// TIA Portal V20 export
DATA_BLOCK "instFB_AxisCtrl"   // DB
TITLE = Axis Control instance DB
{ S7_Optimized_Access := 'TRUE' }
// iDB for FB_AxisCtrl — per-axis MC_Power/Home/Reset for SCARA 4-joint kinematic
// stored: InstanceOfName FB_AxisCtrl, InstanceOfType FB
"FB_AxisCtrl"
BEGIN
END_DATA_BLOCK
